            IF (_MessageLevel > E_MessageType.eMessageError)
            THEN
              _stMsg.eType                              := E_MessageType.eMessageInfo;
              _stMsg.eSubdevice                         := e_Subdevice.Application_Init;
              _stMsg.iErrorNumber                       := 0;
              _stMsg.sText                              := concat(TO_STRING(E_INSTANCE.SENDER_BUFFER_INFEED), ': init');
              f_MessageSet(_stMsg);

              _stMsg.eType                              := E_MessageType.eMessageInfo;
              _stMsg.eSubdevice                         := e_Subdevice.Application_Init;
              _stMsg.iErrorNumber                       := 0;
              _stMsg.sText                              := concat(TO_STRING(_eState), ': ');
              f_MessageSet(_stMsg);
            END_IF
            GVL_MSG.ApplicationMessageCtrl.Cmd          := E_MESSAGE_CTRL.MSG_CTRL_WRITE;
        END_CASE
    END_CASE
END_CASE
//-----------------------------------------------------------------------------------------------------------------
//-----------------------------------------------------------------------------------------------------------------
Init                                                    := _eState;
END_METHOD

PROPERTY InstanceCtrl : REFERENCE TO ARRAY[1..MAX_PROCESS] OF ST_INSTANCE_CTRL
SET
_InstanceCtrl REF= InstanceCtrl;
END_SET
END_PROPERTY

PROPERTY InstanceState : REFERENCE TO ARRAY[1..MAX_PROCESS] OF ST_INSTANCE_STATE
SET
_InstanceState REF= InstanceState;
END_SET
END_PROPERTY

PROPERTY ListControl : REFERENCE TO ST_LIST_CTRL
SET
_InfeedListCtrl REF= ListControl;
END_SET
END_PROPERTY

METHOD ListData   : E_PROGRESS  // simulates data entry from transfersystem into BUFFER_INFEED linked list
VAR_INPUT
  Execute         : BOOL;
END_VAR
VAR_INST
  _nBit,
  _nExp           : BYTE;
  _nMod           : UINT := 5;

  _eStateProgress,
  _eRslt          : E_PROGRESS;

  _ProcessData    : ST_PROCESS_DATA;

  _nMinListCount  : UDINT := 1;
  _nWaitcountLast,
  _nWaitCount     : UDINT;

  _tMsg           : ST_Message;
END_VAR
//---------------------------------------------------------------------------------------
IF NOT Execute
THEN
  _eStateProgress             := E_PROGRESS.PROGRESS_INIT;
END_IF
//---------------------------------------------------------------------------------------
IF NOT Check() 
THEN 
	ListData                    := E_PROGRESS.PROGRESS_ERROR; 
	RETURN; 
END_IF
//---------------------------------------------------------------------------------------
_tMsg.eDevice                 := _stMsg.eDevice; 
//---------------------------------------------------------------------------------------
//---------------------------------------------------------------------------------------
CASE _eStateProgress
OF
   E_PROGRESS.PROGRESS_INIT:
    IF Execute
    THEN
      IF (_InfeedListState.Count < 1)
      THEN
        _ListDataWaitCounterOld := _ListDataWaitCounter;
        _ListDataWaitCounter    := 0;

        _InfeedListCtrl.Cmd     := E_LIST_CTRL.LIST_CTRL_NULL;
        _eStateProgress         :=  E_PROGRESS.PROGRESS_BUSY;

        IF (_MessageLevel > E_MessageType.eMessageError)
        THEN
          _tMsg.eType         := E_MessageType.eMessageInfo;
          _tMsg.eSubdevice    := e_Subdevice.Application;
          _tMsg.iErrorNumber  := _nTicketCount;
          _tMsg.sText         := concat('ListData.TicketCount: ', TO_STRING(_nTicketCount));
          f_MessageSet(_tMsg);
        END_IF
      ELSE
        _ListDataWaitCounter    := _ListDataWaitCounter + 1;
      END_IF
    END_IF

  E_PROGRESS.PROGRESS_BUSY:
    CASE _nLoadCase
    OF
      0:  // fully loaded
        _eStateProgress       := E_PROGRESS.PROGRESS_CHECK;
        _nLoadCaseOld         := _nLoadCase;

        IF (_MessageLevel > E_MessageType.eMessageError)
        THEN
          _tMsg.eType         := E_MessageType.eMessageInfo;
          _tMsg.eSubdevice    := e_Subdevice.Application;
          _tMsg.iErrorNumber  := _nLoadCase;
          _tMsg.sText         := concat('ListData.Progress: ', TO_STRING(_eStateProgress));
          _tMsg.sText         := concat(_tMsg.sText, ': LoadCase: ');
          _tMsg.sText         := concat(_tMsg.sText, TO_STRING(_nLoadCase));
   
          f_MessageSet(_tMsg);
        END_IF


      1:  // static bits
        _eStateProgress       := E_PROGRESS.PROGRESS_PREPARE;
        _nLoadCaseOld         := _nLoadCase;

        IF (_MessageLevel > E_MessageType.eMessageError)
        THEN
          _tMsg.eType          := E_MessageType.eMessageInfo;
          _tMsg.eSubdevice     := e_Subdevice.Application;
          _tMsg.iErrorNumber   := _nLoadCase;
          _tMsg.sText         := concat('ListData.Progress: ', TO_STRING(_eStateProgress));
          _tMsg.sText         := concat(_tMsg.sText, ': LoadCase: ');
          _tMsg.sText         := concat(_tMsg.sText, TO_STRING(_nLoadCase));
          f_MessageSet(_tMsg);
        END_IF


      2:  // incrementing bits
        _eStateProgress       := E_PROGRESS.PROGRESS_STARTUP;
        _nLoadCaseOld         := _nLoadCase;

        IF (_MessageLevel > E_MessageType.eMessageError)
        THEN
          _tMsg.eType          := E_MessageType.eMessageInfo;
          _tMsg.eSubdevice     := e_Subdevice.Application;
          _tMsg.iErrorNumber   := _nLoadCase;
          _tMsg.sText         := concat('ListData.Progress: ', TO_STRING(_eStateProgress));
          _tMsg.sText         := concat(_tMsg.sText, ': LoadCase: ');
          _tMsg.sText         := concat(_tMsg.sText, TO_STRING(_nLoadCase));
          f_MessageSet(_tMsg);
        END_IF


      99:
        _eStateProgress       := E_PROGRESS.PROGRESS_WORKING;
        _ProcessData.wTarget  := 0;

        IF (_MessageLevel > E_MessageType.eMessageError)
        THEN
          _tMsg.eType          := E_MessageType.eMessageInfo;
          _tMsg.eSubdevice     := e_Subdevice.Application;
          _tMsg.iErrorNumber   := _nLoadCase;
          _tMsg.sText          := concat(TO_STRING(_eState), ': _ProcessData.wTarget: ');
          _tMsg.sText          := concat(_stMsg.sText, f_BitsToString(_ProcessData.wTarget));
          f_MessageSet(_tMsg);
        END_IF
        _nLoadCase            := _nLoadCaseOld;

    ELSE
        _eStateProgress       := E_PROGRESS.PROGRESS_STARTUP;
    END_CASE
    _nWaitCount               := 0; 
END_CASE
//---------------------------------------------------------------------------------------
//---------------------------------------------------------------------------------------
CASE _eStateProgress
OF
  E_PROGRESS.PROGRESS_PREPARE:
    _eStateProgress           := E_PROGRESS.PROGRESS_WORKING;
    _nExp                     := TO_BYTE(_InstanceState[E_INSTANCE.INFEED].StationCount);
    _ProcessData.wTarget      := f_To_T_Process(_nExp);

    IF (_nTicketCount MOD _nMod = 0)
    THEN
      _nBit                   := SEL((_nBit>_nExp), _nBit+1, 0);
      _ProcessData.wTarget    := f_BitDel(_ProcessData.wTarget, _nBit);
    END_IF
    IF (_nTicketCount MOD (8) = 0)
    THEN
      _nBit                   := 1;
      _ProcessData.wTarget    := f_BitDel(_ProcessData.wTarget, _nBit);
    END_IF
    IF (_nTicketCount MOD (16) = 0)
    THEN
      _nBit                   := 2;
      _ProcessData.wTarget    := f_BitDel(_ProcessData.wTarget, _nBit);
    END_IF
    IF (_nTicketCount MOD (24) = 0)
    THEN
      _nBit                   := 3;
      _ProcessData.wTarget    := f_BitDel(_ProcessData.wTarget, _nBit);
    END_IF
    IF (_nTicketCount MOD (32) = 0)
    THEN
      _nBit                   := 4;
      _ProcessData.wTarget    := f_BitDel(_ProcessData.wTarget, _nBit);
    END_IF
    IF (_nTicketCount MOD (40) = 0)
    THEN
      _nBit                   := 5;
      _ProcessData.wTarget    := f_BitDel(_ProcessData.wTarget, _nBit);
    END_IF
    IF (_nTicketCount MOD (48) = 0)
    THEN
      _nBit                   := 6;
      _ProcessData.wTarget    := f_BitDel(_ProcessData.wTarget, _nBit);
    END_IF
    IF (_nTicketCount MOD (60) = 0)
    THEN
      _nBit                   := 7;
      _ProcessData.wTarget    := f_BitDel(_ProcessData.wTarget, _nBit);
    END_IF
    IF (_nTicketCount MOD (72) = 0)
    THEN
      _nBit                   := 8;
      _ProcessData.wTarget    := f_BitDel(_ProcessData.wTarget, _nBit);
    END_IF
    IF (_nTicketCount MOD (84) = 0)
    THEN
      _nBit                   := 9;
      _ProcessData.wTarget    := f_BitDel(_ProcessData.wTarget, _nBit);
    END_IF
    IF (_nTicketCount MOD (96) = 0)
    THEN
      _nBit                   := 10;
      _ProcessData.wTarget    := f_BitDel(_ProcessData.wTarget, _nBit);
    END_IF
    IF (_nTicketCount MOD (108) = 0)
    THEN
      _nBit                   := 11;
      _ProcessData.wTarget    := f_BitDel(_ProcessData.wTarget, _nBit);
    END_IF
    IF (_MessageLevel > E_MessageType.eMessageError)
    THEN
      _tMsg.eType             := E_MessageType.eMessageInfo;
      _tMsg.eSubdevice        := e_Subdevice.Application;
      _tMsg.iErrorNumber      := _nLoadCase;
      _tMsg.sText             := concat('ListData.Progress: ', TO_STRING(_eState));
      _tMsg.sText             := concat(_tMsg.sText, ': _ProcessData.wTarget: ');
      _tMsg.sText             := concat(_tMsg.sText, f_BitsToString(_ProcessData.wTarget));
      f_MessageSet(_tMsg);
    END_IF
END_CASE
//---------------------------------------------------------------------------------------
//---------------------------------------------------------------------------------------
CASE _eStateProgress
OF
  E_PROGRESS.PROGRESS_STARTUP:
    _eStateProgress           := E_PROGRESS.PROGRESS_WORKING;
    _nExp                     := TO_BYTE(_InstanceState[E_INSTANCE.INFEED].StationCount);
    _ProcessData.wTarget      := f_To_T_Process(_nExp);

    IF (_nTicketCount MOD _nMod = 0)
    THEN
      _nBit                   := SEL((_nBit>_nExp), _nBit+1, 0);
      _ProcessData.wTarget    := f_BitDel(_ProcessData.wTarget, _nBit);
    END_IF
    IF (_MessageLevel > E_MessageType.eMessageError)
    THEN
      _tMsg.eType             := E_MessageType.eMessageInfo;
      _tMsg.eSubdevice        := e_Subdevice.Application;
      _tMsg.iErrorNumber      := _nLoadCase;
      _tMsg.sText             := concat('ListData.Progress: ', TO_STRING(_eState));
      _tMsg.sText             := concat(_tMsg.sText, ': _ProcessData.wTarget: ');
      _tMsg.sText             := concat(_tMsg.sText, f_BitsToString(_ProcessData.wTarget));
      f_MessageSet(_tMsg);
    END_IF
END_CASE
//---------------------------------------------------------------------------------------
//---------------------------------------------------------------------------------------
CASE _eStateProgress
OF
  E_PROGRESS.PROGRESS_CHECK:
    _eStateProgress           := E_PROGRESS.PROGRESS_WORKING;
    _nExp                     := TO_BYTE(_InstanceState[E_INSTANCE.INFEED].StationCount);
    _ProcessData.wTarget      := f_To_T_Process(_nExp);

    _InfeedListDataInput.ProcessData  := _ProcessData;

    IF (_MessageLevel > E_MessageType.eMessageError)
    THEN
      _tMsg.eType             := E_MessageType.eMessageInfo;
      _tMsg.eSubdevice        := e_Subdevice.Application;
      _tMsg.iErrorNumber      := _nLoadCase;
      _tMsg.sText             := concat('ListData.Progress: ', TO_STRING(_eState));
      _tMsg.sText             := concat(_tMsg.sText, ': _ProcessData.wTarget: ');
      _tMsg.sText             := concat(_tMsg.sText, f_BitsToString(_ProcessData.wTarget));
      f_MessageSet(_tMsg);
    END_IF
    IF (_MessageLevel > E_MessageType.eMessageEmpty)
    THEN
      _tMsg.eType             := E_MessageType.eMessageInfo;
      _tMsg.eDevice           := e_Device.Metrics;
      _tMsg.eSubdevice        := e_Subdevice.Application;
      _tMsg.iErrorNumber      := _nLoadCase;
      _tMsg.sText             := concat('ListData.Progress: ', TO_STRING(_eState));
      _tMsg.sText             := concat(_tMsg.sText, ': _ProcessData.wTarget: ');
      _tMsg.sText             := concat(_tMsg.sText, f_BitsToString(_ProcessData.wTarget));
      f_MessageSet(_tMsg);
    END_IF
END_CASE
//---------------------------------------------------------------------------------------
//---------------------------------------------------------------------------------------
CASE _eStateProgress
OF
  E_PROGRESS.PROGRESS_WORKING:
    _InfeedListDataInput.ProcessData            := _ProcessData;
    _InfeedListDataInput.ProcessData.nProcessId := E_INSTANCE.BUFFER_INFEED;
    _InfeedListCtrl.Cmd                         := E_LIST_CTRL.LIST_CTRL_ADD_TAIL;

    IF (_InfeedListState.State = E_LIST_STATE.LIST_STATE_ADD_TAIL + E_PROGRESS.PROGRESS_ERROR)
    THEN
      _eStateProgress         := E_PROGRESS.PROGRESS_ERROR;

      _tMsg.eType             := E_MessageType.eMessageError;
      _tMsg.eSubdevice        := e_Subdevice.Application;
      _tMsg.iErrorNumber      := _nLoadCase;
      _tMsg.sText             := concat('AddTail: ', TO_STRING(E_INSTANCE.BUFFER_INFEED));
      _tMsg.sText             := concat(_tMsg.sText, ': ');
      _tMsg.sText             := concat(_tMsg.sText, TO_STRING(_eStateProgress));
      f_MessageSet(_tMsg);

    ELSIF(_InfeedListState.State = E_LIST_STATE.LIST_STATE_ADD_TAIL + E_PROGRESS.PROGRESS_DONE)
    THEN
       _nTicketCount          := _nTicketCount + 1;
      _eStateProgress         := E_PROGRESS.PROGRESS_OCCUPIED;
 
     IF (_MessageLevel > E_MessageType.eMessageError)
      THEN
        _tMsg.eType           := E_MessageType.eMessageInfo;
        _tMsg.eSubdevice      := e_Subdevice.Application;
        _tMsg.iErrorNumber    := _nLoadCase;
        _tMsg.sText           := concat('AddTail: ', TO_STRING(E_INSTANCE.BUFFER_INFEED));
        _tMsg.sText           := concat(_tMsg.sText, ': ');
        _tMsg.sText           := concat(_tMsg.sText, TO_STRING(E_PROGRESS.PROGRESS_DONE));
        f_MessageSet(_tMsg);
      END_IF
    END_IF
END_CASE
//---------------------------------------------------------------------------------------
//---------------------------------------------------------------------------------------
CASE _eStateProgress
OF
  E_PROGRESS.PROGRESS_OCCUPIED:
    _InfeedListCtrl.Cmd       := E_LIST_CTRL.LIST_CTRL_NULL;
    _nWaitCount               := _nWaitCount + 1;
    _eStateProgress           :=  E_PROGRESS.PROGRESS_DONE;
END_CASE

ListData                      := _eStateProgress;
END_METHOD

PROPERTY ListInputData : REFERENCE TO ST_LIST_NODE_DATA
SET
_InfeedListDataInput REF= ListInputData;
END_SET
END_PROPERTY

PROPERTY ListState : REFERENCE TO ST_LIST_STATE
SET
_InfeedListState REF= ListState;
END_SET
END_PROPERTY

PROPERTY MessageLevel : e_MessageType
GET
MessageLevel := _MessageLevel;
END_GET
SET
_MessageLevel := MessageLevel;
END_SET
END_PROPERTY

METHOD Proceed : E_PROGRESS
VAR_INPUT
  Execute     : BOOL;
END_VAR
VAR_INST
  _nErrorId               : UDINT;
  _eRslt,
  _eState                 : E_PROGRESS;

  _eInst                  : E_INSTANCE;
  _TransportState         : E_XTS_TRANSPORT_STATE;
  _bDbg : BOOL;
END_VAR
//-----------------------------------------------------------------------------
IF NOT Execute 
THEN 
	_eState                                   := E_PROGRESS.PROGRESS_INIT; 
END_IF 
//-----------------------------------------------------------------------------
IF NOT Check() 
THEN 
	Proceed                                   := E_PROGRESS.PROGRESS_ERROR; 
	RETURN; 
END_IF
//-----------------------------------------------------------------------------
//-----------------------------------------------------------------------------
CASE _eState
OF
  E_PROGRESS.PROGRESS_INIT:
    IF Execute
    THEN
      _nErrorId                             := 0;

      IF (_XtsTransportState.GroupInfo.AxisCountEnabled = _XtsTransportState.XpuInfo.nExpectedAxisCount) AND
         (_XtsTransportState.GroupInfo.AxisCount        = _XtsTransportState.XpuInfo.nExpectedAxisCount)
      THEN
        IF NOT (_Ctrl.Variant = E_APP_VARIANT.VARIANT_INVALID)
        THEN
          _eState                           := E_PROGRESS.PROGRESS_BUSY;
          _XtsTransportCtrl.Cmd             := E_XTS_TRANSPORT_CTRL.CMD_NULL;
  
          IF (_MessageLevel > E_MessageType.eMessageError)
          THEN
            _stMsg.eType                    := E_MessageType.eMessageInfo;
            _stMsg.eSubdevice               := e_Subdevice.Application_Proceed;
            _stMsg.iErrorNumber             := 0;
            _stMsg.sText                    := concat(TO_STRING(_eState), ': ');
            f_MessageSet(_stMsg);
          END_IF
        END_IF
      ELSE
        _nErrorId                           := _eState;

        _eState                             := E_PROGRESS.PROGRESS_ERROR;

        _stMsg.eType                        := E_MessageType.eMessageError;
        _stMsg.eSubdevice                   := e_Subdevice.Application_Proceed;
        _stMsg.iErrorNumber                 := _nErrorId;
        _stMsg.sText                        := concat(TO_STRING(_eState), ': ');
        _stMsg.sText                        := concat(_stMsg.sText, TO_STRING(_XtsTransportState.GroupInfo.AxisCountEnabled));
        _stMsg.sText                        := concat(_stMsg.sText, ' / ');
        _stMsg.sText                        := concat(_stMsg.sText, TO_STRING(_XtsTransportState.GroupInfo.AxisCount));
        _stMsg.sText                        := concat(_stMsg.sText, ' CaGroup Axis mismatch');
        f_MessageSet(_stMsg);
      END_IF
    END_IF


  E_PROGRESS.PROGRESS_BUSY:
    _XtsTransportCtrl.Cmd                   := E_XTS_TRANSPORT_CTRL.CMD_TRANSPORT_RESTART;

    IF (_XtsTransportState.State = E_XTS_TRANSPORT_STATE.TRANSPORT_RESTART + E_PROGRESS.PROGRESS_ERROR)
    THEN
      _eState                               := E_PROGRESS.PROGRESS_ERROR;
      _TransportState                       := _XtsTransportState.State MOD E_PROGRESS.PROGRESS_ERROR;

      _stMsg.eType                          := E_MessageType.eMessageError;
      _stMsg.eSubdevice                     := e_Subdevice.Application_Proceed;
      _stMsg.iErrorNumber                   := _nErrorId;
      _stMsg.sText                          := concat(TO_STRING(_eState), ': ');
      _stMsg.sText                          := concat(_stMsg.sText, TO_STRING(_TransportState));
      f_MessageSet(_stMsg);

    ELSIF (_XtsTransportState.State = E_XTS_TRANSPORT_STATE.TRANSPORT_RESTART + E_PROGRESS.PROGRESS_DONE)
    THEN
      _eState                               := E_PROGRESS.PROGRESS_WORKING;
      _TransportState                       := _XtsTransportState.State MOD E_PROGRESS.PROGRESS_DONE;
      _eRslt                                := ListData(FALSE);

      IF (_MessageLevel > E_MessageType.eMessageError)
      THEN
        _stMsg.eType                        := E_MessageType.eMessageInfo;
        _stMsg.eSubdevice                   := e_Subdevice.Application_Proceed;
        _stMsg.iErrorNumber                 := 0;
        _stMsg.sText                        := concat(TO_STRING(_eState), ': ');
        _stMsg.sText                        := concat(_stMsg.sText, TO_STRING(_TransportState));
        f_MessageSet(_stMsg);
      END_IF
    END_IF

END_CASE
//-----------------------------------------------------------------------------
//-----------------------------------------------------------------------------
CASE _eState
OF
  E_PROGRESS.PROGRESS_WORKING:

    FOR _eInst := E_INSTANCE.PROCESS_CONDUCTOR TO E_INSTANCE.SENDER_BUFFER_INFEED
    DO
      // handshakes to instances: 
      // - deconstruct this for your own implementation
      CASE _InstanceState[_eInst].State
      OF
        E_INSTANCE_STATE.DISABLED:
          CASE _InstanceState[_eInst].Progress
          OF
            E_PROGRESS.PROGRESS_BUSY:
              IF NOT (_eInst = E_INSTANCE.INFEED)
              THEN
                _InstanceCtrl[_eInst].Cmd   := E_INSTANCE_CMD.ENABLE;
              ELSE
                _eRslt                      := ListData(TRUE);

                IF (_eRslt = E_PROGRESS.PROGRESS_DONE)
                THEN
                  _InstanceCtrl[_eInst].Cmd := E_INSTANCE_CMD.ENABLE;
                END_IF
              END_IF
          END_CASE
      
        E_INSTANCE_STATE.ENABLED:
          CASE _InstanceState[_eInst].Progress
          OF
            E_PROGRESS.PROGRESS_OCCUPIED:
              _InstanceCtrl[_eInst].Cmd     := E_INSTANCE_CMD.PROCEED;
          END_CASE
      
        E_INSTANCE_STATE.WORKING:
          CASE _InstanceState[_eInst].Progress
          OF
            E_PROGRESS.PROGRESS_BUSY:
              _tonProcess [_eInst]
                              (IN           := FALSE, 
                               PT           := _tProcess[_eInst]);

              IF (_eInst > E_INSTANCE.OUTFEED_ROBOT_R2) OR
                 (_eInst < E_INSTANCE.OUTFEED_ROBOT_R1) OR
                 (_bSingleOutput) OR
                 NOT (_Ctrl.Variant = E_APP_VARIANT.VARIANT_OUTPUT_24)
              THEN
                _InstanceCtrl[_eInst].Cmd   := E_INSTANCE_CMD.WORK;
              ELSE
                IF (_InstanceState[E_INSTANCE.OUTFEED_ROBOT_R1].State = 
                    _InstanceState[E_INSTANCE.OUTFEED_ROBOT_R2].State )
                THEN
                  // in this example the outfeed instances are working in sync
                  _InstanceCtrl[_eInst].Cmd := E_INSTANCE_CMD.WORK;
                ELSE
                  CASE _InstanceState[E_INSTANCE.OUTFEED_ROBOT_R2].State
                  OF
                    E_INSTANCE_STATE.ENABLED:
                      // in case R2 is empty --> unload R1
                      _InstanceCtrl[E_INSTANCE.OUTFEED_ROBOT_R1].Cmd := E_INSTANCE_CMD.WORK;
                  END_CASE
                END_IF
              END_IF
      
      
            E_PROGRESS.PROGRESS_CHECK:
              _tonProcess [_eInst]
                              (IN           := TRUE, 
                               PT           := _tProcess[_eInst]);
      
              IF _tonProcess [_eInst].Q
              THEN
                _InstanceCtrl[_eInst].Cmd   := E_INSTANCE_CMD.FINISH;
              END_IF
          END_CASE


        E_INSTANCE_STATE.FINISH:
          CASE _InstanceState[_eInst].Progress
          OF
            E_PROGRESS.PROGRESS_BUSY:
              _InstanceCtrl[_eInst].Cmd     := E_INSTANCE_CMD.FINISH;

            E_PROGRESS.PROGRESS_OCCUPIED:
              _InstanceCtrl[_eInst].Cmd     := E_INSTANCE_CMD.PROCEED;

            e_progress.PROGRESS_DONE:
              _InstanceCtrl[_eInst].Cmd     := E_INSTANCE_CMD.FINISH;
              _eRslt                        := ListData(FALSE);
          END_CASE
        END_CASE
    END_FOR
END_CASE
//-----------------------------------------------------------------------------
//-----------------------------------------------------------------------------

Proceed                                     := _eState;
END_METHOD

PROPERTY State : REFERENCE TO ST_APP_STATE
SET
_State ref= State;
END_SET
END_PROPERTY

METHOD Work : E_PROGRESS  // cyclic handshakes with timers, 
                          // this procedure you have to build for your own application. 
                          // This simulated work method is here 
                          // because it was convinient for me to do so
VAR_INPUT
  Execute                 : BOOL;
END_VAR
VAR_INST
  _nErrorId               : UDINT;
  _eRslt,
  _eState                 : E_PROGRESS;

  _eInst                  : E_INSTANCE;
  _bDbg : BOOL;

  _TransportState         : E_XTS_TRANSPORT_STATE;
  _JobResult              : E_PROGRESS;

  _tonListData            : Tc2_Standard.TON;
  _tListDataIntervall     : time := t#20ms;
END_VAR
//-----------------------------------------------------------------------------
IF NOT Execute 
THEN 
	_eState                                   := E_PROGRESS.PROGRESS_INIT; 
END_IF 
//-----------------------------------------------------------------------------
IF NOT Check() 
THEN 
	Work                                      := E_PROGRESS.PROGRESS_ERROR; 
	RETURN; 
END_IF
//-----------------------------------------------------------------------------
//-----------------------------------------------------------------------------
CASE _eState
OF
  E_PROGRESS.PROGRESS_INIT:
    IF Execute
    THEN
      _nErrorId                             := 0;

      IF (_XtsTransportState.GroupInfo.AxisCountEnabled = _XtsTransportState.XpuInfo.nExpectedAxisCount) AND
         (_XtsTransportState.GroupInfo.AxisCount        = _XtsTransportState.XpuInfo.nExpectedAxisCount)
      THEN
        IF NOT (_Ctrl.Variant = E_APP_VARIANT.VARIANT_INVALID)
        THEN
          _eState                           := E_PROGRESS.PROGRESS_BUSY;
          _XtsTransportCtrl.Cmd             := E_XTS_TRANSPORT_CTRL.CMD_NULL;
          _eRslt                            := Clear(FALSE);
  
          IF (_MessageLevel > E_MessageType.eMessageError)
          THEN
            _stMsg.eType                    := E_MessageType.eMessageInfo;
            _stMsg.eSubdevice               := e_Subdevice.Application_Work;
            _stMsg.iErrorNumber             := 0;
            _stMsg.sText                    := concat(TO_STRING(_eState), ': ');
            f_MessageSet(_stMsg);
          END_IF
        END_IF
      ELSE
        _nErrorId                           := _XtsTransportState.GroupInfo.AxisCountEnabled;
        _eState                             := E_PROGRESS.PROGRESS_ERROR;

        _stMsg.eType                        := E_MessageType.eMessageError;
        _stMsg.eSubdevice                   := e_Subdevice.Application_Work;
        _stMsg.iErrorNumber                 := _nErrorId;
        _stMsg.sText                        := concat(TO_STRING(_eState), ': ');
        _stMsg.sText                        := concat(_stMsg.sText, TO_STRING(_XtsTransportState.GroupInfo.AxisCountEnabled));
        _stMsg.sText                        := concat(_stMsg.sText, ' / ');
        _stMsg.sText                        := concat(_stMsg.sText, TO_STRING(_XtsTransportState.GroupInfo.AxisCount));
        _stMsg.sText                        := concat(_stMsg.sText, ' CaGroup Axis mismatch');
        f_MessageSet(_stMsg);
      END_IF
    END_IF

  E_PROGRESS.PROGRESS_BUSY:
    _eRslt                                  := Clear(TRUE);

    IF (_eRslt = E_PROGRESS.PROGRESS_DONE)
    THEN
      _XtsTransportCtrl.Cmd     := E_XTS_TRANSPORT_CTRL.CMD_TRANSPORT_START;
  
      IF (_XtsTransportState.State = E_XTS_TRANSPORT_STATE.TRANSPORT_START + E_PROGRESS.PROGRESS_ERROR)
      THEN
        _eState                             := E_PROGRESS.PROGRESS_ERROR;
        _TransportState                     := _XtsTransportState.State MOD E_PROGRESS.PROGRESS_ERROR;

        _stMsg.eType                        := E_MessageType.eMessageError;
        _stMsg.eSubdevice                   := e_Subdevice.Application_Work;
        _stMsg.iErrorNumber                 := _nErrorId;
        _stMsg.sText                        := concat(TO_STRING(_eState), ': ');
        _stMsg.sText                        := concat(_stMsg.sText, TO_STRING(_TransportState));
        f_MessageSet(_stMsg);
  
      ELSIF (_XtsTransportState.State = E_XTS_TRANSPORT_STATE.TRANSPORT_START + E_PROGRESS.PROGRESS_DONE)
      THEN
        _eState                             := E_PROGRESS.PROGRESS_PREPARE;
        _TransportState                     := _XtsTransportState.State MOD E_PROGRESS.PROGRESS_DONE;

        IF (_MessageLevel > E_MessageType.eMessageError)
        THEN
          _stMsg.eType                      := E_MessageType.eMessageInfo;
          _stMsg.eSubdevice                 := e_Subdevice.Application_Work;
          _stMsg.iErrorNumber               := 0;
          _stMsg.sText                      := concat(TO_STRING(_eState), ': ');
          _stMsg.sText                      := concat(_stMsg.sText, TO_STRING(_TransportState));
          f_MessageSet(_stMsg);
        END_IF
      END_IF
    END_IF

  E_PROGRESS.PROGRESS_PREPARE:
    _eRslt                                  := ListData(FALSE);
    IF (_eRslt = E_PROGRESS.PROGRESS_INIT)
    THEN
      _eState                               := E_PROGRESS.PROGRESS_STARTUP;
      _InfeedListCtrl.Cmd                   := e_list_ctrl.LIST_CTRL_NULL;

      _InfeedListDataInput.ProcessData.wTarget    := f_To_T_Process(TO_BYTE(_InstanceState[E_INSTANCE.INFEED].StationCount));
      _InfeedListDataInput.ProcessData.nProcessId := E_INSTANCE.SENDER_BUFFER_INFEED;
    END_IF     


  E_PROGRESS.PROGRESS_STARTUP:  // SENDER_BUFFER_INFEED sends the first batch of movers to BUFFER_INFEED
                                //  - after sending the first batch 
                                //    --> the transfersystem (ListData) may start writing entries into BUFFER_INFEED
    CASE _InstanceState[E_INSTANCE.SENDER_BUFFER_INFEED].State
    OF
    E_INSTANCE_STATE.DISABLED:

      CASE _InstanceState[E_INSTANCE.SENDER_BUFFER_INFEED].Progress
      OF
      E_PROGRESS.PROGRESS_BUSY:
        _eState                             := E_PROGRESS.PROGRESS_CHECK;
        _InfeedListCtrl.Cmd                 := e_list_ctrl.LIST_CTRL_ADD_TAIL;

        IF (_MessageLevel > E_MessageType.eMessageError)
        THEN
          _stMsg.eType                      := E_MessageType.eMessageInfo;
          _stMsg.eSubdevice                 := e_Subdevice.Application_Work;
          _stMsg.iErrorNumber               := 0;
          _stMsg.sText                      := concat(TO_STRING(_eState), ': ');
          _stMsg.sText                      := concat(_stMsg.sText, TO_STRING(e_Subdevice.Process_LinkedList_AddTail));
          f_MessageSet(_stMsg);
        END_IF
      END_CASE
    END_CASE
END_CASE
//-----------------------------------------------------------------------------
//-----------------------------------------------------------------------------
CASE _eState
OF
  E_PROGRESS.PROGRESS_CHECK:
    IF (_InfeedListState.State = e_list_state.LIST_STATE_ADD_TAIL + e_progress.PROGRESS_DONE)
    THEN
      _eState                                         := E_PROGRESS.PROGRESS_OCCUPIED;
      _InfeedListCtrl.Cmd                             := e_list_ctrl.LIST_CTRL_NULL;
      _InstanceCtrl[E_INSTANCE.PROCESS_CONDUCTOR].Cmd := E_INSTANCE_CMD.ENABLE;
      _InstanceCtrl[E_INSTANCE.BUFFER_INFEED].Cmd     := E_INSTANCE_CMD.ENABLE;


    ELSIF (_InfeedListState.State = e_list_state.LIST_STATE_ADD_TAIL + e_progress.PROGRESS_ERROR)
    THEN
      _eState                               := E_PROGRESS.PROGRESS_ERROR;
    END_IF 
END_CASE
//-----------------------------------------------------------------------------
//-----------------------------------------------------------------------------
CASE _eState
OF
  E_PROGRESS.PROGRESS_OCCUPIED:
    _eState                     := E_PROGRESS.PROGRESS_WORKING;

    IF (_MessageLevel > E_MessageType.eMessageError)
    THEN
      _stMsg.eType                          := E_MessageType.eMessageInfo;
      _stMsg.eSubdevice                     := e_Subdevice.Application_Work;
      _stMsg.iErrorNumber                   := 0;
      _stMsg.sText                          := concat(TO_STRING(_eState), ': ');
      f_MessageSet(_stMsg);
    END_IF
END_CASE
//-----------------------------------------------------------------------------
//-----------------------------------------------------------------------------
CASE _eState
OF
  E_PROGRESS.PROGRESS_WORKING:
    FOR _eInst := E_INSTANCE.PROCESS_CONDUCTOR TO E_INSTANCE.SENDER_BUFFER_INFEED
    DO
      // handshakes to instances: 
      // - deconstruct this for your own implementation
      CASE _InstanceState[_eInst].State
      OF
        E_INSTANCE_STATE.DISABLED:
          CASE _InstanceState[_eInst].Progress
          OF
            E_PROGRESS.PROGRESS_BUSY:
            CASE _eInst
            OF
              e_instance.PROCESS_CONDUCTOR:

                CASE _InstanceState[e_instance.BUFFER_INFEED].State
                OF
                  E_INSTANCE_STATE.DETECTION:
                    _eRslt                  := ListData(FALSE);
                    _tonListData( IN        := FALSE,
                                  PT        := _tListDataIntervall);
                    IF NOT _bTicketCountOverride
                    THEN
                      IF (_nTicketCount < _nTicketCountEnd+1)
                      THEN
                        _InstanceCtrl[e_instance.PROCESS_CONDUCTOR].Cmd := E_INSTANCE_CMD.ENABLE;
                      END_IF
                    ELSE
                      _InstanceCtrl[e_instance.PROCESS_CONDUCTOR].Cmd   := E_INSTANCE_CMD.ENABLE;
                    END_IF
                END_CASE
            ELSE
                _InstanceCtrl[_eInst].Cmd := E_INSTANCE_CMD.ENABLE;
            END_CASE
          END_CASE
      
        E_INSTANCE_STATE.ENABLED:
          CASE _InstanceState[_eInst].Progress
          OF
            E_PROGRESS.PROGRESS_OCCUPIED:
              _InstanceCtrl[_eInst].Cmd     := E_INSTANCE_CMD.PROCEED;
          END_CASE

        E_INSTANCE_STATE.WORKING:
          CASE _InstanceState[_eInst].Progress
          OF
            E_PROGRESS.PROGRESS_BUSY:
              _tonProcess [_eInst]
                              (IN           := FALSE, 
                               PT           := _tProcess[_eInst]);


              IF (_eInst > E_INSTANCE.OUTFEED_ROBOT_R2) OR
                 (_eInst < E_INSTANCE.OUTFEED_ROBOT_R1) OR
                 (_bSingleOutput) OR
                 NOT (_Ctrl.Variant = E_APP_VARIANT.VARIANT_OUTPUT_24)
              THEN
                _InstanceCtrl[_eInst].Cmd   := E_INSTANCE_CMD.WORK;
              ELSE
                IF (_InstanceState[E_INSTANCE.OUTFEED_ROBOT_R1].State = 
                    _InstanceState[E_INSTANCE.OUTFEED_ROBOT_R2].State )
                THEN
                  // in this example the outfeed instances are working in sync
                  _InstanceCtrl[_eInst].Cmd := E_INSTANCE_CMD.WORK;
                END_IF
              END_IF
      
      
            E_PROGRESS.PROGRESS_CHECK:
              _tonProcess [_eInst]
                              (IN           := TRUE, 
                               PT           := _tProcess[_eInst]);
      
              IF _tonProcess [_eInst].Q
              THEN
                _InstanceCtrl[_eInst].Cmd   := E_INSTANCE_CMD.FINISH;
              END_IF
          END_CASE


        E_INSTANCE_STATE.FINISH:
          CASE _InstanceState[_eInst].Progress
          OF
            E_PROGRESS.PROGRESS_BUSY:
              _tonProcess [_eInst]
                              (IN           := FALSE, 
                               PT           := _tProcess[_eInst]);

              _InstanceCtrl[_eInst].Cmd     := E_INSTANCE_CMD.FINISH;

            E_PROGRESS.PROGRESS_OCCUPIED:
              _InstanceCtrl[_eInst].Cmd     := E_INSTANCE_CMD.PROCEED;

            E_PROGRESS.PROGRESS_DONE:
              _tonListData(IN               := TRUE,
                           PT               := _tListDataIntervall);
              IF (_tonListData.Q)
              THEN
                _eRslt                        := ListData(_bRunListData);
                IF (_eRslt = E_PROGRESS.PROGRESS_DONE)
                THEN
                  _InstanceCtrl[_eInst].Cmd   := E_INSTANCE_CMD.FINISH;
                END_IF
              END_IF
          END_CASE
        END_CASE
    END_FOR
END_CASE
//-----------------------------------------------------------------------------
//-----------------------------------------------------------------------------
Work                                        := _eState;
END_METHOD

PROPERTY WriteTimeVariant : bool
GET
WriteTimeVariant := _bWriteTimeVariant;
END_GET
SET
_bWriteTimeVariant := WriteTimeVariant;
END_SET
END_PROPERTY

PROPERTY XtsTransportCtrl : REFERENCE TO ST_XTS_TRANSPORT_CTRL
SET
_XtsTransportCtrl REF= XtsTransportCtrl;
END_SET
END_PROPERTY

PROPERTY XtsTransportState : REFERENCE TO ST_XTS_TRANSPORT_STATE
SET
_XtsTransportState REF= XtsTransportState;
END_SET
END_PROPERTY

END_FUNCTION_BLOCK

// ---- MSG/f_MessageSet.TcPOU
FUNCTION f_MessageSet : BOOL
VAR_INPUT
  stMessage     : ST_Message;
END_VAR
VAR
  _uiIndex      : UINT;
  _MainDevice   : e_Device;
  _nModRes      : UDINT;     // residual after modulo
END_VAR

stMessage.tTime                     := GVL_MSG.sLocalTime;

// why here? so all calls to this function may stay the same
_nModRes                            := stMessage.eDevice MOD e_Device.General;
_MainDevice                         := stMessage.eDevice - _nModRes;

CASE _MainDevice
OF
  e_device.DataProduct:
    // this is your data, if you choose to use this message system
    FOR _uiIndex := 1 TO GVL_MSG.MAX_MESSAGE
    DO
      IF (GVL_MSG.ProductMessages[_uiIndex].eType = e_MessageType.eMessageEmpty)
      THEN
        GVL_MSG.ProductMessages[_uiIndex]      := stMessage;
        GVL_MSG.MessageProductIndex            := _uiIndex;
        EXIT;
      END_IF
    END_FOR
  
    IF (stMessage.eType = E_MessageType.eMessageError)
    THEN
      // in case of error: increment counter
      GVL_MSG.MessageProductError     := GVL_MSG.MessageProductError + 1;
    END_IF


  e_Device.Process,
  e_Device.Application:
    FOR _uiIndex := 1 TO GVL_MSG.MAX_MESSAGE
    DO
      IF (GVL_MSG.ApplicationMessages[_uiIndex].eType = e_MessageType.eMessageEmpty)
      THEN
        GVL_MSG.ApplicationMessages[_uiIndex]  := stMessage;    // yes, we grab global values directly, only here
        GVL_MSG.MessageApplicationIndex        := _uiIndex;
        EXIT;
      END_IF
    END_FOR
    IF (stMessage.eType = E_MessageType.eMessageError)
    THEN
      // in case of error: increment counter
      GVL_MSG.MessageApplicationError := GVL_MSG.MessageApplicationError + 1;
    END_IF

  e_Device.Metrics:
    FOR _uiIndex := 1 TO GVL_MSG.MAX_MESSAGE
    DO
      IF (GVL_MSG.MetricsMessages[_uiIndex].eType = e_MessageType.eMessageEmpty)
      THEN
        GVL_MSG.MetricsMessages[_uiIndex]  := stMessage;    // yes, we grab global values directly, only here
        GVL_MSG.MessageMetricsIndex        := _uiIndex;
        EXIT;
      END_IF
    END_FOR
    IF (stMessage.eType = E_MessageType.eMessageError)
    THEN
      // in case of error: increment counter
      GVL_MSG.MessageMetricsError := GVL_MSG.MessageMetricsError + 1;
    END_IF

ELSE
  FOR _uiIndex := 1 TO GVL_MSG.MAX_MESSAGE
  DO
    IF (GVL_MSG.TransportMessages[_uiIndex].eType = e_MessageType.eMessageEmpty)
    THEN
      GVL_MSG.TransportMessages[_uiIndex]      := stMessage;
      GVL_MSG.MessageTransportIndex            := _uiIndex;
      EXIT;
    END_IF
  END_FOR

  IF (stMessage.eType = E_MessageType.eMessageError)
  THEN
    // in case of error: increment counter
    GVL_MSG.MessageTransportError := GVL_MSG.MessageTransportError + 1;
  END_IF
END_CASE

END_FUNCTION

// ---- XTS/_types/f_BitSet.TcPOU
FUNCTION f_BitSet : T_PROCESS
VAR_INPUT
  inVal   : T_PROCESS;
  bitNo   : DINT;
END_VAR
VAR
  wConst  : T_PROCESS := 1;
END_VAR

f_BitSet := inVal OR SHL( wConst,TO_SINT(bitNo) MOD TO_INT(SIZEOF(T_PROCESS)*8) );

END_FUNCTION

// ---- XTS/_types/f_BitGet.TcPOU
FUNCTION f_BitGet : BOOL
VAR_INPUT
  inVal   : T_PROCESS;
  bitNo   : DINT;
END_VAR
VAR
  wConst : T_PROCESS := 1;
END_VAR

IF ( inVal AND SHL( wConst,TO_SINT(bitNo) MOD TO_INT(SIZEOF(T_PROCESS)*8) ) ) > 0
THEN
  f_BitGet := TRUE;
ELSE
  f_BitGet := FALSE;
END_IF

END_FUNCTION

// ---- APPLICATION/_types/f_To_T_Process.TcPOU
FUNCTION f_To_T_Process : T_process
VAR_INPUT
  nExp              : BYTE;
END_VAR
VAR
  rVal              : LREAL;
  nTmp              : ULINT; 
  wTmp              : T_PROCESS;
END_VAR

rVal   := TO_LREAL(SEL(nExp > SIZEOF(T_PROCESS)*8, nExp, SIZEOF(T_PROCESS)*8));
nTmp   := TO_ULINT(EXPT(2,rVal)-1);

memcpy(ADR(wtmp), ADR(ntmp), SIZEOF(wtmp));

f_To_T_Process      := wtmp;

END_FUNCTION

// ---- XTS/_types/f_BitDel.TcPOU
FUNCTION f_BitDel : T_PROCESS
VAR_INPUT
  inVal   : T_PROCESS;
  bitNo   : DINT;
END_VAR
VAR
  wConst : T_PROCESS := 1;
END_VAR

IF ( inVal AND SHL( wConst,TO_SINT(bitNo) MOD TO_INT(SIZEOF(T_PROCESS)*8) ) ) > 0 THEN
  f_BitDel := inVal XOR (SHL( wConst,TO_SINT(bitNo) MOD TO_INT(SIZEOF(T_PROCESS)*8) ));
ELSE
  f_BitDel := inVal;
END_IF

END_FUNCTION

// ---- MSG/fb_MessageDataCtrl.TcPOU
FUNCTION_BLOCK fb_MessageDataCtrl EXTENDS fb_MessageData
VAR
  _stCtrl       : REFERENCE TO ST_MESSAGE_CTRL;
  _stState      : REFERENCE TO ST_MESSAGE_STATE;

  _eCmd,
  _eCmdOld      : E_MESSAGE_CTRL;

  _eResult,
  _eJobResult   : E_PROGRESS;

  _eState       : E_MESSAGE_STATE;

END_VAR

//-----------------------------------------------------------------------------
// check pointers
//-----------------------------------------------------------------------------
IF NOT Check()
THEN
  _eResult                      := E_PROGRESS.PROGRESS_ERROR;
  RETURN;
END_IF
//-----------------------------------------------------------------------------
// check date
// new message file for a new day
//-----------------------------------------------------------------------------
IF (FolderDate(_dtLocalTime) <> _sFolderDate)
THEN
  _bFileCreated                 := FALSE;
END_IF
//-----------------------------------------------------------------------------
//----------------------------------------------------------------------------- 
// copy to local for debug
_eCmd                         := _stCtrl.Cmd;

// cyclic check for command change
// get state for cmd
IF (_eCmd <> _eCmdOld)
THEN
  // get matching sdtate for Ctrl.Cmd
  _eState                     := Cmd(_eCmd);
  _eCmdOld                    := _eCmd;
END_IF


CASE _eResult
OF
  E_PROGRESS.PROGRESS_INVALID:
    _stState.State            := E_MESSAGE_STATE.MSG_STATE_NULL;

  E_PROGRESS.PROGRESS_ERROR:
    _stState.State            := _eState + E_PROGRESS.PROGRESS_ERROR;

  E_PROGRESS.PROGRESS_DONE:
    _stState.State            := _eState + E_PROGRESS.PROGRESS_DONE;

ELSE
  // work in progress
  // update progress for extern use
  _stState.State              := _eState + _eResult;

  CASE _eState
  OF
    E_MESSAGE_STATE.MSG_STATE_INIT:
      _eResult                := BuildFolder(TRUE);


    E_MESSAGE_STATE.MSG_STATE_IDLE:
      IF (_nMsgIndex < GVL_MSG.MAX_MESSAGE - GVL_MSG.MAX_MESSAGE/10)
      THEN
        _eResult              := E_PROGRESS.PROGRESS_WORKING;
      ELSE
        _eResult              := E_PROGRESS.PROGRESS_DONE;
        _nMsgIndex            := 0;
        // copy from attached list to local
        memcpy(ADR(_aWriteList), _pMsgList, SIZEOF(_aWriteList));
        // clear attached list
        memset(_pMsgList, 0, SIZEOF(_aWriteList));
      END_IF


    E_MESSAGE_STATE.MSG_STATE_WRITE:
      _eResult                := BuildFileData(TRUE);

  ELSE
      _eResult               := E_PROGRESS.PROGRESS_INVALID;
  END_CASE
END_CASE

METHOD BuildFileData : e_progress
VAR_INPUT
  Execute     : BOOL;
END_VAR
VAR_INST
  _nErrorId   : UDINT;
  _eState,
  _eRes       : E_PROGRESS;
  _eFlow      : E_MESSAGE_FLOW;

  _nStringLength  : UINT;
END_VAR
//-----------------------------------------------------------------------------
IF NOT Execute 
THEN
  _eRes                           := WriteData(FALSE);
  _eRes                           := BuildFolder(FALSE);
	_eState                         := E_PROGRESS.PROGRESS_INIT; 
END_IF 
//-----------------------------------------------------------------------------
IF NOT Check() 
THEN 
	BuildFileData                   := E_PROGRESS.PROGRESS_ERROR; 
	RETURN; 
END_IF
//-----------------------------------------------------------------------------
//-----------------------------------------------------------------------------
CASE _eState
OF
  E_PROGRESS.PROGRESS_INIT:
    IF Execute
    THEN
      _nErrorId                   := 0;
      _iStart 	                  := 1;
      _iEnd 		                  := SEL((_nMsgIndex > GVL_MSG.MAX_MESSAGE-1),
                                          _nMsgIndex,
                                          GVL_MSG.MAX_MESSAGE);

      memset(ADR(_sWriteData),0,SIZEOF(_sWriteData));

      IF (_sFolderDate <> FolderDate(_dtLocalTime))
      THEN
        _eState                   := E_PROGRESS.PROGRESS_PREPARE;
      ELSE
        _eState                   := E_PROGRESS.PROGRESS_BUSY;
        _eFlow                    := E_MESSAGE_FLOW.MSG_FLOW_LINE_START;
      END_IF
    END_IF
END_CASE
//-----------------------------------------------------------------------------
//-----------------------------------------------------------------------------
CASE _eState
OF
  E_PROGRESS.PROGRESS_PREPARE:
    _eRes                         := BuildFolder(TRUE);
    CASE _eRes
    OF
      E_PROGRESS.PROGRESS_DONE:
      _eState                     := E_PROGRESS.PROGRESS_BUSY;
      _eFlow                      := E_MESSAGE_FLOW.MSG_FLOW_LINE_START;

      E_PROGRESS.PROGRESS_ERROR:
      _eState                     := E_PROGRESS.PROGRESS_ERROR;
    END_CASE
END_CASE
//-----------------------------------------------------------------------------
//-----------------------------------------------------------------------------
CASE _eState
OF
  E_PROGRESS.PROGRESS_BUSY:
  CASE _eFlow
  OF
    E_MESSAGE_FLOW.MSG_FLOW_LINE_START:
      _eRes                       := BuildFolder(FALSE);
      _nErrIndex                  := 0; // rise and shine, all quarrels erased but not forgotten
      _nMsgIndex                  := 0;
  
      // copy from attached list to local
      memcpy(ADR(_aWriteList), _pMsgList, SIZEOF(_aWriteList));
  
      // clear attached list
      memset(_pMsgList, 0, SIZEOF(_aWriteList));


      _eFlow                      := E_MESSAGE_FLOW.MSG_FLOW_LINE_BUILD;
      _iCount                     := _iStart;
  END_CASE
  CASE _eFlow
  OF
    E_MESSAGE_FLOW.MSG_FLOW_LINE_BUILD:
      _eFlow                      := E_MESSAGE_FLOW.MSG_FLOW_LINE_CHECK;
      IF (_aWriteList[_iCount].eType > E_MessageType.eMessageEmpty)
      THEN
        _sTmp                     := TO_STRING(_aWriteList[_iCount].eType);
        _sTmp                     := Tc2_Standard.CONCAT(_sTmp, _sTab);
        _sTmp                     := Tc2_Standard.CONCAT(_sTmp, _aWriteList[_iCount].tTime);
        _sTmp                     := Tc2_Standard.CONCAT(_sTmp, _sTab);
        _sTmp                     := Tc2_Standard.CONCAT(_sTmp, Device_To_String(_aWriteList[_iCount].eDevice));
        _sTmp                     := Tc2_Standard.CONCAT(_sTmp, _sTab);
        _sTmp                     := Tc2_Standard.CONCAT(_sTmp, TO_STRING(_aWriteList[_iCount].eSubdevice));
        _sTmp                     := Tc2_Standard.CONCAT(_sTmp, _sTab);
        _sTmp                     := Tc2_Standard.CONCAT(_sTmp, TO_STRING(_aWriteList[_iCount].iErrorNumber));
        _sTmp                     := Tc2_Standard.CONCAT(_sTmp, _sTab);
        _sTmp                     := Tc2_Standard.CONCAT(_sTmp, _aWriteList[_iCount].sText);
        _sTmp                     := Tc2_Standard.CONCAT(_sTmp, _sNewLine);
        Builder(ADR(_sTmp), ADR(_sWriteData), StringLen(ADR(_sTmp)));
      END_IF
      _iCount                     := _iCount + 1;
  END_CASE
  CASE _eFlow
  OF
    E_MESSAGE_FLOW.MSG_FLOW_LINE_CHECK:
    IF NOT (_iCount > _iEnd)
    THEN
      _eFlow                      := E_MESSAGE_FLOW.MSG_FLOW_LINE_BUILD;
    ELSE
      _eState                     := E_PROGRESS.PROGRESS_WORKING;
      _eFlow                      := E_MESSAGE_FLOW.MSG_FLOW_WRITE_FILE_BUSY;
    END_IF
  END_CASE
END_CASE
//-----------------------------------------------------------------------------
//-----------------------------------------------------------------------------
CASE _eState
OF
  E_PROGRESS.PROGRESS_WORKING:
  CASE _eFlow
  OF
    E_MESSAGE_FLOW.MSG_FLOW_WRITE_FILE_BUSY:
      _nStringLength              := StringLen(ADR(_sWriteData));
      IF NOT (_nStringLength > 1)
      THEN
        _eState                   := E_PROGRESS.PROGRESS_DONE; 
       _eFlow                     := E_MESSAGE_FLOW.MSG_FLOW_WRITE_FILE_DONE;
      ELSE
        _eFlow                    := E_MESSAGE_FLOW.MSG_FLOW_WRITE_FILE_END;
        _eRes                     := WriteData(FALSE);
      END_IF
  END_CASE
  CASE _eFlow
  OF
    E_MESSAGE_FLOW.MSG_FLOW_WRITE_FILE_END:
      _eRes                       := WriteData(TRUE);

      IF (_eRes = E_PROGRESS.PROGRESS_ERROR)
      THEN
        _eState                   := E_PROGRESS.PROGRESS_ERROR;

      ELSIF (_eRes = E_PROGRESS.PROGRESS_DONE)
      THEN
        _eState                   := E_PROGRESS.PROGRESS_DONE;
        _eFlow                    := E_MESSAGE_FLOW.MSG_FLOW_WRITE_FILE_DONE;
        _eRes                     := WriteData(FALSE);
      END_IF
  END_CASE
END_CASE
//-----------------------------------------------------------------------------
//-----------------------------------------------------------------------------

BuildFileData                     := _eState;
END_METHOD

METHOD BuildFolder : e_progress
VAR_INPUT
  Execute           : BOOL;
END_VAR
VAR_INST
  _nErrorId   : UDINT;
  _eState     : E_PROGRESS;
  _eFlow      : E_MESSAGE_FLOW;
END_VAR
//-----------------------------------------------------------------------------
IF NOT Execute 
THEN 
	_eState                       := E_PROGRESS.PROGRESS_INIT; 
END_IF 
//-----------------------------------------------------------------------------
IF NOT Check() 
THEN 
	BuildFolder                   := E_PROGRESS.PROGRESS_ERROR; 
	RETURN; 
END_IF
//-----------------------------------------------------------------------------
//-----------------------------------------------------------------------------
CASE _eState
OF
  E_PROGRESS.PROGRESS_INIT:
    IF Execute
    THEN
      _nErrorId                 := 0;
      _bFileCreated             := FALSE;

      _sFolderDate              := FolderDate(_dtLocalTime);
      _eState                   := E_PROGRESS.PROGRESS_BUSY;
      _eFlow                    := E_MESSAGE_FLOW.MSG_FLOW_ROOT;
    END_IF
END_CASE
//-----------------------------------------------------------------------------
//-----------------------------------------------------------------------------
CASE _eState
OF
  E_PROGRESS.PROGRESS_BUSY:
  CASE _eFlow
  OF
    E_MESSAGE_FLOW.MSG_FLOW_ROOT:
      _eFlow                    := E_MESSAGE_FLOW.MSG_FLOW_ROOT_CREATE;
      _fbCreateDir.sPathName    := left(_pDirRoot^,len(_pDirRoot^)-1);
      _fbCreateDir(
              bExecute	        := FALSE);
    
    E_MESSAGE_FLOW.MSG_FLOW_ROOT_CREATE:
      (* create root folder *)
      _fbCreateDir(
              bExecute	        := TRUE);
      IF _fbCreateDir.bBusy
      THEN
        _eFlow                  := E_MESSAGE_FLOW.MSG_FLOW_ROOT_CREATE_BUSY;
      END_IF
    
    E_MESSAGE_FLOW.MSG_FLOW_ROOT_CREATE_BUSY:
      _fbCreateDir(
              bExecute	        := TRUE);
      IF NOT _fbCreateDir.bBusy
      THEN
        _eState                 := E_PROGRESS.PROGRESS_PREPARE;
        _eFlow                  := E_MESSAGE_FLOW.MSG_FLOW_FOLDER;
      END_IF
  END_CASE
END_CASE
//-----------------------------------------------------------------------------
//-----------------------------------------------------------------------------
CASE _eState
OF
  E_PROGRESS.PROGRESS_PREPARE:
  CASE _eFlow
  OF
    E_MESSAGE_FLOW.MSG_FLOW_FOLDER:
      _eFlow                    := E_MESSAGE_FLOW.MSG_FLOW_FOLDER_CREATE;
      _sFolderDate              := FolderDate(_dtLocalTime);
      _fbCreateDir.sPathName    := concat(_pDirRoot^, _sFolderDate);
      _fbCreateDir(
              bExecute	        := FALSE);
  
    E_MESSAGE_FLOW.MSG_FLOW_FOLDER_CREATE:
      (* create active folder *)
      _fbCreateDir(
              bExecute	        := TRUE);
      IF _fbCreateDir.bBusy
      THEN
        _eFlow                  := E_MESSAGE_FLOW.MSG_FLOW_FOLDER_CREATE_BUSY;
      END_IF
    
    E_MESSAGE_FLOW.MSG_FLOW_FOLDER_CREATE_BUSY:
      _fbCreateDir(
              bExecute	        := TRUE);
      IF NOT _fbCreateDir.bBusy
      THEN
        _eState                 := E_PROGRESS.PROGRESS_CHECK;
        _eFlow                  := E_MESSAGE_FLOW.MSG_FLOW_FILE_CREATE_DONE;
        _fbCreateDir(
                bExecute	      := FALSE);
      END_IF
  END_CASE
END_CASE
//-----------------------------------------------------------------------------
//-----------------------------------------------------------------------------
CASE _eState
OF
  E_PROGRESS.PROGRESS_CHECK:
  CASE _eFlow
  OF
    E_MESSAGE_FLOW.MSG_FLOW_FILE_CREATE_DONE:
      _eState                   := E_PROGRESS.PROGRESS_DONE;
      _bFileCreated             := TRUE;

      // build complete file path
      _sTmp                     := concat(concat(_pFileRoot^, _sFolderDate),'.txt');
      _sTmp                     := concat('\', _sTmp);
      _sFilename                := concat(_fbCreateDir.sPathName, _sTmp);
  END_CASE
END_CASE

BuildFolder                     := _eState;
END_METHOD

METHOD Check : BOOL
VAR_INPUT
END_VAR

IF NOT __ISVALIDREF(_stCtrl)
THEN
  _eCheck       := E_MESSAGE_CHECK.MSG_CHECK_INVALID_POINTER_CTRL;
  RETURN;
END_IF

IF NOT __ISVALIDREF(_stState)
THEN
  _eCheck       := E_MESSAGE_CHECK.MSG_CHECK_INVALID_POINTER_STATE;
  RETURN;
END_IF
//-----------------------------------------------------------------
//-----------------------------------------------------------------
IF NOT (_dtLocalTime <> 0)
THEN
  _eCheck       := E_MESSAGE_CHECK.MSG_CHECK_INVALID_POINTER_TIME;
  RETURN;
END_IF

IF NOT (_pMsgList <> 0)
THEN
  _eCheck       := E_MESSAGE_CHECK.MSG_CHECK_INVALID_POINTER_LIST;
  RETURN;
END_IF

IF NOT (_pFileRoot <> 0)
THEN
  _eCheck       := E_MESSAGE_CHECK.MSG_CHECK_INVALID_POINTER_ROOT_FILE;
  RETURN;
END_IF

IF NOT (_pDirRoot <> 0)
THEN
  _eCheck       := E_MESSAGE_CHECK.MSG_CHECK_INVALID_POINTER_ROOT_DIR;
  RETURN;
END_IF

IF NOT __ISVALIDREF(_nMsgIndex)
THEN
  _eCheck       := E_MESSAGE_CHECK.MSG_CHECK_INVALID_POINTER_MSG_IDX;
  RETURN;
END_IF

IF NOT __ISVALIDREF(_nErrIndex)
THEN
  _eCheck       := E_MESSAGE_CHECK.MSG_CHECK_INVALID_POINTER_ERR_IDX;
  RETURN;
END_IF


_eCheck         := E_MESSAGE_CHECK.MSG_CHECK_DONE;
Check           := TRUE;
END_METHOD

METHOD Cmd : e_message_state
VAR_INPUT
  Command     : e_message_ctrl;
END_VAR


CASE Command
OF
  E_MESSAGE_CTRL.MSG_CTRL_NULL:
    _eResult                    := E_PROGRESS.PROGRESS_INVALID;
    Cmd                         := E_MESSAGE_STATE.MSG_STATE_NULL;

  E_MESSAGE_CTRL.MSG_CTRL_INIT:
    _eResult                    := BuildFolder(FALSE);
    Cmd                         := E_MESSAGE_STATE.MSG_STATE_INIT;

  E_MESSAGE_CTRL.MSG_CTRL_IDLE:
    _eResult                    := BuildFileData(FALSE);
    Cmd                         := E_MESSAGE_STATE.MSG_STATE_IDLE;

  E_MESSAGE_CTRL.MSG_CTRL_WRITE:
    _eResult                    := BuildFileData(FALSE);
    Cmd                         := E_MESSAGE_STATE.MSG_STATE_WRITE;
    IF (_nMsgIndex = 0)
    THEN
       // go back to sleep
      _eResult                := E_PROGRESS.PROGRESS_DONE;
    END_IF
ELSE
    //_eResult                    := E_PROGRESS.PROGRESS_ERROR;
    Cmd                         := E_MESSAGE_STATE.MSG_STATE_NULL;
END_CASE
END_METHOD

PROPERTY Ctrl : REFERENCE to ST_MESSAGE_CTRL
SET
_stCtrl ref= Ctrl;
END_SET
END_PROPERTY

PROPERTY FileCreated : bool
GET
FileCreated := _bFileCreated;
END_GET
END_PROPERTY

PROPERTY State : REFERENCE TO ST_MESSAGE_STATE
SET
_stState ref= State;
END_SET
END_PROPERTY

END_FUNCTION_BLOCK

// ---- MSG/fb_MessageData.TcPOU
FUNCTION_BLOCK ABSTRACT fb_MessageData IMPLEMENTS I_MessageData
VAR CONSTANT
{attribute 'hide'}
  STR_LEN       : UDINT := 524_288;
END_VAR
VAR
  _eCheck       : E_MESSAGE_CHECK;            // pointer check state

  _pFileRoot    : POINTER TO STRING(255);     // you decide (example in GVL_MSG.LOG_FILE)
  _pDirRoot     : POINTER TO STRING(255);     // see GVL_MSG.LOG_DIR

  _nMsgIndex    : REFERENCE TO UINT;          // Hypnos IS the only one in the village, if there are more you need more villages
  _nErrIndex    : REFERENCE TO UINT;          // Thanatos, Hypnos stern and more serious brother

  _dtLocalTime  : POINTER TO DT;
  _pMsgList     : POINTER TO ARRAY[1..GVL_MSG.MAX_MESSAGE] OF ST_Message; // attach your list here

	_rtrigReset   : Tc2_Standard.R_TRIG;
	_aWriteList   : ARRAY[1..GVL_MSG.MAX_MESSAGE] OF ST_Message;
	_sWriteData   : STRING(STR_LEN);
	_sNewLine     : STRING := '$N';
	_sTab         : STRING := '$T';
	_iCount, 
	_iStart, 
	_iEnd         : UINT;

	_fbCreateDir  : Tc2_System.FB_CreateDir;
	_sTmp         : STRING(256);
	_sFilename    : STRING(256);
	_sFolderDate  : STRING;
	_bFileCreated : BOOL;

	_fbFileOpen   : Tc2_System.FB_FileOpen;
	_fbFileWrite  : Tc2_System.FB_FileWrite;
	_fbFileClose  : Tc2_System.FB_FileClose;
END_VAR

METHOD Builder : BOOL // string concat for length > 255
VAR_INPUT
  pInString   : POINTER TO STRING;
  pOutString  : POINTER TO STRING(STR_LEN);
  Length      : UINT;
END_VAR
VAR
  Counter     : UDINT;
  pInWork     : POINTER TO BYTE;
  pOutWork    : POINTER TO BYTE;
END_VAR
pOutWork := pOutString;
pInWork := pInString;
Counter := 0;

(*check termination*)
WHILE (pOutWork^ <> 0) AND
      (Counter < STR_LEN+1)
DO
  Counter := Counter + 1;
  pOutWork := pOutWork + 1;
END_WHILE

(* append only if data fits into output *)
IF (Counter + Length < STR_LEN+1)
THEN

  (* append data *)
  FOR Counter := 1 TO Length
  DO
    pOutWork^ := pInWork^;
    pOutWork := pOutWork + 1;
    pInWork := pInWork + 1;
  END_FOR

  (* terminate *)
  pOutWork := pOutWork + 1;
  pOutWork^ := 0;
END_IF
END_METHOD

METHOD Check : BOOL
VAR_INPUT
END_VAR

IF NOT (_dtLocalTime <> 0)
THEN
  _eCheck       := E_MESSAGE_CHECK.MSG_CHECK_INVALID_POINTER_TIME;
  RETURN;
END_IF

IF NOT (_pMsgList <> 0)
THEN
  _eCheck       := E_MESSAGE_CHECK.MSG_CHECK_INVALID_POINTER_LIST;
  RETURN;
END_IF

IF NOT (_pFileRoot <> 0)
THEN
  _eCheck       := E_MESSAGE_CHECK.MSG_CHECK_INVALID_POINTER_ROOT_FILE;
  RETURN;
END_IF

IF NOT (_pDirRoot <> 0)
THEN
  _eCheck       := E_MESSAGE_CHECK.MSG_CHECK_INVALID_POINTER_ROOT_DIR;
  RETURN;
END_IF

IF NOT __ISVALIDREF(_nMsgIndex)
THEN
  _eCheck       := E_MESSAGE_CHECK.MSG_CHECK_INVALID_POINTER_MSG_IDX;
  RETURN;
END_IF

IF NOT __ISVALIDREF(_nErrIndex)
THEN
  _eCheck       := E_MESSAGE_CHECK.MSG_CHECK_INVALID_POINTER_ERR_IDX;
  RETURN;
END_IF


_eCheck         := E_MESSAGE_CHECK.MSG_CHECK_DONE;
Check           := TRUE;
END_METHOD

METHOD Device_to_String : string
VAR_INPUT
  eMsgDevice    : e_Device;
END_VAR
VAR
  sId                 : STRING := '_ID_';
  nId                 : UDINT;
END_VAR
IF (eMsgDevice < e_device.General)
THEN
  // below general case
  nId := TO_UDINT(eMsgDevice);
  sId := concat(sId, TO_STRING(nId));

  Device_to_String := concat(TO_STRING(eMsgDevice), sId);

ELSE
  IF (eMsgDevice >= e_Device.DataProduct)
  THEN
    nId := eMsgDevice MOD e_Device.DataProduct;
    sId := concat(sId, TO_STRING(nId));
 
    Device_to_String := concat(TO_STRING(e_Device.DataProduct), sId);

  ELSIF (eMsgDevice >= e_Device.Application)
  THEN
    nId := eMsgDevice MOD e_Device.Application;
    sId := concat(sId, TO_STRING(nId));
 
    Device_to_String := concat(TO_STRING(e_Device.Application), sId);

  ELSIF (eMsgDevice >= e_Device.Process)
  THEN
    nId := eMsgDevice MOD e_Device.Process;
    sId := concat(sId, TO_STRING(nId));
 
    Device_to_String := concat(TO_STRING(e_Device.Process), sId);

  ELSIF (eMsgDevice >= e_Device.Metrics)
  THEN
    nId := eMsgDevice MOD e_Device.Metrics;
    sId := concat(sId, TO_STRING(nId));
 
    Device_to_String := concat(TO_STRING(e_device.Metrics), sId);

  ELSIF (eMsgDevice >= e_device.XfcAxis)
  THEN
    nId := eMsgDevice MOD e_device.XfcAxis;
    sId := concat(sId, TO_STRING(nId));
 
    Device_to_String := concat(TO_STRING(e_device.XfcAxis), sId);

  ELSIF (eMsgDevice >= e_device.Axis)
  THEN
    nId := eMsgDevice MOD e_device.Axis;
    sId := concat(sId, TO_STRING(nId));
 
    Device_to_String := concat(TO_STRING(e_device.Axis), sId);

  ELSIF (eMsgDevice >= e_device.NciChannelCtrl)
  THEN
    nId := eMsgDevice MOD e_device.NciChannelCtrl;
    sId := concat(sId, TO_STRING(nId));
 
    Device_to_String := concat(TO_STRING(e_device.NciChannelCtrl), sId);

  ELSIF (eMsgDevice >= e_device.NciChannel)
  THEN
    nId := eMsgDevice MOD e_device.NciChannel;
    sId := concat(sId, TO_STRING(nId));
 
    Device_to_String := concat(TO_STRING(e_device.NciChannel), sId);

  ELSIF (eMsgDevice >= e_Device.Camming)
  THEN
    nId := eMsgDevice MOD e_Device.Camming;
    sId := concat(sId, TO_STRING(nId));
 
    Device_to_String := concat(TO_STRING(e_device.Camming), sId);

  ELSIF (eMsgDevice >= e_Device.XtsStation)
  THEN
    nId := eMsgDevice MOD e_Device.XtsStation;
    sId := concat(sId, TO_STRING(nId));
 
    Device_to_String := concat(TO_STRING(e_device.XtsStation), sId);

  ELSIF (eMsgDevice >= e_Device.XfcTouchProbe)
  THEN
    nId := eMsgDevice MOD e_Device.XfcTouchProbe;
    sId := concat(sId, TO_STRING(nId));
 
    Device_to_String := concat(TO_STRING(e_device.XfcTouchProbe), sId);

  ELSIF (eMsgDevice >= e_Device.XfcTriggerBox)
  THEN
    nId := eMsgDevice MOD e_Device.XfcTriggerBox;
    sId := concat(sId, TO_STRING(nId));
 
    Device_to_String := concat(TO_STRING(e_device.XfcTriggerBox), sId);

  ELSIF (eMsgDevice >= e_Device.XtsTransportUnit)
  THEN
    nId := eMsgDevice MOD e_Device.XtsTransportUnit;
    sId := concat(sId, TO_STRING(nId));
 
    Device_to_String := concat(TO_STRING(e_device.XtsTransportUnit), sId);

  ELSIF (eMsgDevice >= e_Device.MoverCtrl)
  THEN
    nId := eMsgDevice MOD e_Device.MoverCtrl;
    sId := concat(sId, TO_STRING(nId));
 
    Device_to_String := concat(TO_STRING(e_device.MoverCtrl), sId);

  ELSIF (eMsgDevice >= e_Device.Mover)
  THEN
    nId := eMsgDevice MOD e_Device.Mover;
    sId := concat(sId, TO_STRING(nId));
 
    Device_to_String := concat(TO_STRING(e_device.Mover), sId);

  ELSIF (eMsgDevice >= e_Device.XpuCtrl)
  THEN
    nId := eMsgDevice MOD e_Device.XpuCtrl;
    sId := concat(sId, TO_STRING(nId));
 
    Device_to_String := concat(TO_STRING(e_device.XpuCtrl), sId);

  ELSIF (eMsgDevice >= e_Device.Xpu)
  THEN
    nId := eMsgDevice MOD e_Device.Xpu;
    sId := concat(sId, TO_STRING(nId));
 
    Device_to_String := concat(TO_STRING(e_device.Xpu), sId);

  ELSIF (eMsgDevice >= e_Device.CaGroup)
  THEN
    nId := eMsgDevice MOD e_Device.CaGroup;
    sId := concat(sId, TO_STRING(nId));
 
    Device_to_String := concat(TO_STRING(e_device.CaGroup), sId);

  ELSIF (eMsgDevice >= e_Device.General)
  THEN
    nId := eMsgDevice MOD e_Device.General;
    sId := concat(sId, TO_STRING(nId));
 
    Device_to_String := concat(TO_STRING(e_device.General), sId);

  ELSE
    Device_to_String := TO_STRING(eMsgDevice);
  END_IF
END_IF
END_METHOD

PROPERTY DirRoot : POINTER to string(255)
SET
_pDirRoot := DirRoot;
END_SET
END_PROPERTY

PROPERTY ErrorIndex : reference to uint
SET
_nErrIndex  REF= ErrorIndex;
END_SET
END_PROPERTY

PROPERTY FileRoot : pointer to string(255)
SET
_pFileRoot := FileRoot;
END_SET
END_PROPERTY

METHOD FolderDate : STRING
VAR_INPUT
	LocalTime   : POINTER TO DT;
END_VAR
VAR
	sTmp        : STRING;
END_VAR
IF NOT (LocalTime <> 0)
THEN
	FolderDate := 'NULL';
	RETURN;
END_IF

sTmp := DT_TO_STRING(LocalTime^);

// cut off #dt literal
sTmp := right(sTmp, len(sTmp)-3);

sTmp := replace(sTmp, '_', 1, 5);
sTmp := replace(sTmp, '_', 1, 8);

sTmp := left(sTmp,10);	// year_month_day

FolderDate := sTmp;
END_METHOD

PROPERTY LocalTime : pointer to DT
SET
_dtLocalTime := LocalTime;
END_SET
END_PROPERTY

PROPERTY MessageIndex : reference to uint
SET
_nMsgIndex   REF= MessageIndex;
END_SET
END_PROPERTY

PROPERTY MsgList : pointer to ARRAY[1..GVL_MSG.MAX_MESSAGE] OF st_message
SET
_pMsgList := MsgList;
END_SET
END_PROPERTY

METHOD StringLen : UINT // 	string length for len > 255
VAR_INPUT
  pInString		: POINTER TO STRING(STR_LEN);
END_VAR
VAR
	Counter			: UINT;
	pInWork			: POINTER TO BYTE;
END_VAR
pInWork := pInString;
Counter := 0;

WHILE (pInWork^ <> 0) AND
			(Counter < STR_LEN)
DO
	Counter := Counter + 1;
	pInWork := pInWork + 1;
END_WHILE

StringLen := Counter;
END_METHOD

METHOD WriteData  : e_progress
VAR_INPUT
  bExecute        : BOOL;
END_VAR
VAR_INST
  _eState         : e_progress;
  _bError         : BOOL;
  _nErrorId       : UDINT;
END_VAR
IF NOT bExecute
THEN
  _eState                     := E_PROGRESS.PROGRESS_INIT;
END_IF

CASE _eState 
OF

	E_PROGRESS.PROGRESS_INIT:
    _fbFileOpen(
        sPathName             := _sFilename, 
        nMode                 := FOPEN_MODEAPPEND OR FOPEN_MODEPLUS, 
        ePath                 := PATH_GENERIC, 
        bExecute              := FALSE, 
        tTimeout              := T#5S);

    _fbFileWrite(
        hFile                 := _fbFileOpen.hFile, 
        pWriteBuff            := ADR(_sWriteData), 
        cbWriteLen            := StringLen(ADR(_sWriteData)),
        bExecute              := FALSE, 
        tTimeout              := T#5S);

    _fbFileClose(
        hFile                 := _fbFileOpen.hFile, 
        bExecute              := FALSE, 
        tTimeout              := T#5S);


		IF bExecute
		THEN
      _nErrorId               := 0;
      _eState                 := E_PROGRESS.PROGRESS_BUSY;
		END_IF

	E_PROGRESS.PROGRESS_BUSY:
		_fbFileOpen(bExecute      := TRUE);

    IF _fbFileOpen.bError
    THEN
      _nErrorId               := _fbFileOpen.nErrId;
      _eState                 := E_PROGRESS.PROGRESS_ERROR;

		ELSIF _fbFileOpen.bBusy
		THEN
      _eState                 := E_PROGRESS.PROGRESS_PREPARE;
		END_IF

	E_PROGRESS.PROGRESS_PREPARE:
		_fbFileOpen(bExecute      := TRUE);
		IF NOT _fbFileOpen.bBusy
		THEN
		  _fbFileOpen(bExecute    := FALSE);
      _eState                 := E_PROGRESS.PROGRESS_STARTUP;
		END_IF

	E_PROGRESS.PROGRESS_STARTUP:
    _fbFileWrite(
        hFile                 := _fbFileOpen.hFile, 
        pWriteBuff            := ADR(_sWriteData), 
        cbWriteLen            := StringLen(ADR(_sWriteData)),
        bExecute              := TRUE, 
        tTimeout              := T#5S);

    IF _fbFileWrite.bError
    THEN
      _nErrorId               := _fbFileWrite.nErrId;
      _eState                 := E_PROGRESS.PROGRESS_ERROR;

		ELSIF _fbFileWrite.bBusy
		THEN
      _eState                 := E_PROGRESS.PROGRESS_CHECK;
		END_IF

	E_PROGRESS.PROGRESS_CHECK:
	  _fbFileWrite(bExecute     := TRUE);
		IF NOT _fbFileWrite.bBusy
		THEN
			_fbFileWrite(bExecute   := FALSE);
      _eState                 := E_PROGRESS.PROGRESS_OCCUPIED;
		END_IF

	E_PROGRESS.PROGRESS_OCCUPIED:
    _fbFileClose(
        hFile                 := _fbFileOpen.hFile, 
        bExecute              := TRUE, 
        tTimeout              := T#5S);

    IF _fbFileClose.bError
    THEN
      _nErrorId               := _fbFileClose.nErrId;
      _eState                 := E_PROGRESS.PROGRESS_ERROR;

		ELSIF _fbFileClose.bBusy
		THEN
      _eState                 := E_PROGRESS.PROGRESS_WORKING;
		END_IF

	E_PROGRESS.PROGRESS_WORKING:
    _fbFileClose(bExecute     := TRUE);
		IF NOT _fbFileClose.bBusy
		THEN
			_fbFileClose(bExecute   := FALSE);
      _eState                 := E_PROGRESS.PROGRESS_DONE;
		END_IF

END_CASE
CASE _eState
OF
  E_PROGRESS.PROGRESS_ERROR:
		_fbFileOpen (bExecute     := FALSE);
    _fbFileWrite(bExecute     := FALSE);
    _fbFileClose(bExecute     := FALSE);


END_CASE




WriteData                     := _eState;
END_METHOD

END_FUNCTION_BLOCK

// ---- APPLICATION/MAIN_APP.TcPOU
//---------------------------------------------------------------------------------------------------------------
//
//  HAUD 2025.11.29
//
//  - EXAMPLE, change, adapt, use
//  -----------------------------
//  - processes and top level workflow examples
//  - based on fb_Instance for processes
//  - fb_Application as top level control for starting, stopping, restarting etc..
//---------------------------------------------------------------------------------------------------------------
PROGRAM MAIN_APP
VAR
  eInit                       : E_PROGRESS;   // application startup state info
  nProcess                    : uint;

  stMsg                       : ST_Message;

  _nBufferOutfeedTarget       : ARRAY[1..2] OF E_INSTANCE;
  _nStnFrst                   : UDINT;

  eMsgState                   : e_message_state;
  eMsgProgress                : E_PROGRESS;

END_VAR

//-----------------------------------------------------------------------------------------------------------------
//-----------------------------------------------------------------------------------------------------------------
// check for MAIN.eInit
//  - wait for fb_TransportUnit to be fully started up
//-----------------------------------------------------------------------------------------------------------------
IF NOT (MAIN.eInit = E_PROGRESS.PROGRESS_DONE) 
THEN 
  eInit                                                     := E_PROGRESS.PROGRESS_INVALID; 
  FOR nProcess := E_INSTANCE.BUFFER_INFEED TO MAX_PROCESS
  DO
    GVL_MSG.MessageLevelProcess[nProcess]                   := GVL_MSG.MessageLevel;
  END_FOR
  ApplicationMain.MessageLevel                              := GVL_MSG.MessageLevel;

  RETURN; 
END_IF
//-----------------------------------------------------------------------------------------------------------------
// set MAIN_APP message device identification
//-----------------------------------------------------------------------------------------------------------------
stMsg.eDevice                                               := e_Device.Application;
//-----------------------------------------------------------------------------------------------------------------
//-----------------------------------------------------------------------------------------------------------------
//-----------------------------------------------------------------------------------------------------------------
// /assign dataflow
//-----------------------------------------------------------------------------------------------------------------
//-----------------------------------------------------------------------------------------------------------------
//-----------------------------------------------------------------------------------------------------------------
//-----------------------------------------------------------------------------------------------------------------
//  main application class
//-----------------------------------------------------------------------------------------------------------------

GVL_APPLICATION.ApplicationMain.Ctrl                        REF=  GVL_APPLICATION.AppControl;
GVL_APPLICATION.ApplicationMain.State                       REF=  GVL_APPLICATION.AppState;
GVL_APPLICATION.ApplicationMain.XtsTransportCtrl            REF=  GVL_XTS.XtsTransportCtrl;
GVL_APPLICATION.ApplicationMain.XtsTransportState           REF=  GVL_XTS.XtsTransportState;
GVL_APPLICATION.ApplicationMain.InstanceCtrl                REF=  GVL_APPLICATION.InstanceCtrl;
GVL_APPLICATION.ApplicationMain.InstanceState               REF=  GVL_APPLICATION.InstanceState;
GVL_APPLICATION.ApplicationMain.ListControl                 REF=  GVL_APPLICATION.TicketListControl;
GVL_APPLICATION.ApplicationMain.ListState                   REF=  GVL_APPLICATION.TicketListState;
GVL_APPLICATION.ApplicationMain.ListInputData               REF=  GVL_APPLICATION.TicketListDataInput;


//-----------------------------------------------------------------------------------------------------------------
//-----------------------------------------------------------------------------------------------------------------
//-----------------------------------------------------------------------------------------------------------------
// assign dataflow/
//-----------------------------------------------------------------------------------------------------------------
//-----------------------------------------------------------------------------------------------------------------
//-----------------------------------------------------------------------------------------------------------------
//-----------------------------------------------------------------------------------------------------------------
//  /STARTUP
//
// startup procedure for application
//  - connects processes and XtsStations
//-----------------------------------------------------------------------------------------------------------------
CASE eInit
OF
  E_PROGRESS.PROGRESS_INVALID:                // first cycle startup
    //---------------------------------------------------------------------------------------------------------------
    // first cycle startup
    // - wait for extern to give the command, if we are waiting here MAIN is ready, extern can see that
    //---------------------------------------------------------------------------------------------------------------
    GVL_MSG.ApplicationMessageCtrl.Cmd        := E_MESSAGE_CTRL.MSG_CTRL_NULL;
    eInit                                     := E_PROGRESS.PROGRESS_INIT;

  E_PROGRESS.PROGRESS_INIT:
    //---------------------------------------------------------------------------------------------------------------
    // wait for valid variant
    //---------------------------------------------------------------------------------------------------------------
    CASE GVL_APPLICATION.AppControl.Variant   // this is what you have to decide, two variants are available
    OF
      E_APP_VARIANT.VARIANT_OUTPUT_24:
        eInit                                 := E_PROGRESS.PROGRESS_BUSY;
  
        stMsg.eType                           := E_MessageType.eMessageInfo;
        stMsg.eSubdevice                      := e_Subdevice.General;
        stMsg.iErrorNumber                    := eInit;
        stMsg.sText                           := concat('MAIN_APP.eInit: ', TO_STRING(eInit));
        stMsg.sText                           := concat(stMsg.sText, ': ');
        stMsg.sText                           := concat(stMsg.sText, TO_STRING(E_INSTANCE.OUTFEED_ROBOT_R1));
        stMsg.sText                           := concat(stMsg.sText, ': ');
        stMsg.sText                           := concat(stMsg.sText, TO_STRING(E_INSTANCE.OUTFEED_ROBOT_R2));
        f_MessageSet(stMsg);

      E_APP_VARIANT.VARIANT_OUTPUT_CLAMP:
        eInit                                 := E_PROGRESS.PROGRESS_BUSY;
  
        stMsg.eType                           := E_MessageType.eMessageInfo;
        stMsg.eSubdevice                      := e_Subdevice.General;
        stMsg.iErrorNumber                    := eInit;
        stMsg.sText                           := concat('MAIN_APP.eInit: ', TO_STRING(eInit));
        stMsg.sText                           := concat(stMsg.sText, ': ');
        stMsg.sText                           := concat(stMsg.sText, TO_STRING(E_INSTANCE.OUTFEED_ROBOT_R1));
        f_MessageSet(stMsg);
    END_CASE

  E_PROGRESS.PROGRESS_BUSY:
    //---------------------------------------------------------------------------------------------------------------
    // first cycle startup of all instances
    //---------------------------------------------------------------------------------------------------------------
    GVL_MSG.ApplicationMessageCtrl.Cmd        := E_MESSAGE_CTRL.MSG_CTRL_INIT;
    IF GVL_MSG.ApplicationMessageData.FileCreated
    THEN
      eInit                                   := E_PROGRESS.PROGRESS_STARTUP;
      GVL_MSG.ApplicationMessageCtrl.Cmd      := E_MESSAGE_CTRL.MSG_CTRL_NULL;
    END_IF

  E_PROGRESS.PROGRESS_STARTUP:
    GVL_APPLICATION.AppControl.Cmd            := E_INSTANCE_CMD.INIT;

    IF (GVL_APPLICATION.AppState.State = E_INSTANCE_STATE.INIT + E_PROGRESS.PROGRESS_DONE)
    THEN
      eInit                                   := E_PROGRESS.PROGRESS_PREPARE;
    END_IF

  E_PROGRESS.PROGRESS_PREPARE:
    IF (GVL_APPLICATION.AppState.AppInit = E_PROGRESS.PROGRESS_DONE)
    THEN
      GVL_APPLICATION.TicketListControl.Cmd   := E_LIST_CTRL.LIST_CTRL_NULL; 
      eInit                                   := E_PROGRESS.PROGRESS_CHECK;
    END_IF

  E_PROGRESS.PROGRESS_CHECK:
    GVL_APPLICATION.TicketListControl.Cmd     := E_LIST_CTRL.LIST_CTRL_INIT;

    IF (GVL_APPLICATION.TicketListState.State =  E_LIST_STATE.LIST_STATE_INIT + E_PROGRESS.PROGRESS_DONE)
    THEN
      eInit                                   := E_PROGRESS.PROGRESS_DONE;
    END_IF
END_CASE
//-----------------------------------------------------------------------------------------------------------------
//-----------------------------------------------------------------------------------------------------------------
// STARTUP/
//-----------------------------------------------------------------------------------------------------------------
//-----------------------------------------------------------------------------------------------------------------
//-----------------------------------------------------------------------------------------------------------------
// /cyclic calls
//-----------------------------------------------------------------------------------------------------------------
GVL_APPLICATION.ApplicationMain();

//-----------------------------------------------------------------------------------------------------------------
//############################################################################
// /logging
//############################################################################
GVL_MSG.ApplicationMessageData.Ctrl           REF= GVL_MSG.ApplicationMessageCtrl;
GVL_MSG.ApplicationMessageData.State          REF= GVL_MSG.ApplicationMessageState;

GVL_MSG.ApplicationMessageData.MessageIndex   REF= GVL_MSG.MessageApplicationIndex;
GVL_MSG.ApplicationMessageData.ErrorIndex     REF= GVL_MSG.MessageApplicationError;

GVL_MSG.ApplicationMessageData.DirRoot        :=   ADR(GVL_MSG.LOG_DIR);
GVL_MSG.ApplicationMessageData.FileRoot       :=   ADR(GVL_MSG.LOG_FILE_APP);

GVL_MSG.ApplicationMessageData.MsgList        :=   ADR(GVL_MSG.ApplicationMessages);
GVL_MSG.ApplicationMessageData.LocalTime      :=   ADR(GVL_MSG.dtLocalTime);

GVL_MSG.ApplicationMessageData();

eMsgState                                     := f_GetState   (GVL_MSG.ApplicationMessageState.State);
eMsgProgress                                  := f_GetProgress(GVL_MSG.ApplicationMessageState.State);


CASE eMsgState
OF
  E_MESSAGE_STATE.MSG_STATE_NULL:
    CASE eMsgProgress
    OF
      E_PROGRESS.PROGRESS_INVALID:
        IF (GVL_MSG.MessageApplicationIndex > GVL_MSG.MAX_MESSAGE/100) OR
           (GVL_MSG.MessageApplicationError > 0)
        THEN
          GVL_MSG.ApplicationMessageCtrl.Cmd  := E_MESSAGE_CTRL.MSG_CTRL_WRITE;
        END_IF
    END_CASE

  E_MESSAGE_STATE.MSG_STATE_WRITE:
    CASE eMsgProgress
    OF
      E_PROGRESS.PROGRESS_ERROR,
      E_PROGRESS.PROGRESS_DONE:
        GVL_MSG.ApplicationMessageCtrl.Cmd    := E_MESSAGE_CTRL.MSG_CTRL_NULL;
    END_CASE

ELSE
    CASE eMsgProgress
    OF
      E_PROGRESS.PROGRESS_DONE:
        GVL_MSG.ApplicationMessageCtrl.Cmd    := E_MESSAGE_CTRL.MSG_CTRL_NULL;
    END_CASE
END_CASE
//############################################################################
// logging/
//############################################################################

END_PROGRAM

// ---- MAIN.TcPOU
PROGRAM MAIN
VAR
  eInit     : e_progress := E_PROGRESS.PROGRESS_DONE;

END_VAR

//############################################################################
// Local time; used for timestamps
//############################################################################
GVL_MSG.fbLocalTime(
                    sLocalTime          => GVL_MSG.sLocalTime, 
                    dtLocalTime         => GVL_MSG.dtLocalTime);

END_PROGRAM
